// TIA Portal V19 export
TYPE "udt_LinTranformation"
// stored: Access Published
   STRUCT
      "m" : Real;
      q : Real;
   END_STRUCT;
END_TYPE
